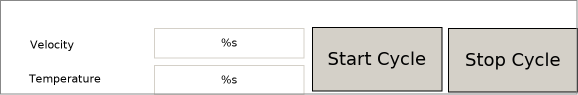
VISUALIZATION BasicHMI  // 578x95
    Textfield (154,28 150x30), "%s", text variable: HMI.Tb_Vel
        OnMouseDown: write HMI.Tb_Vel via VisuDialogs.Numpad
    Label (27,30 120x30), "Velocity"
    Rectangle (312,27 130x64), "Start Cycle"
        tap HMI.Bt_StartCycle
    Label (26,64 120x30), "Temperature"
    Textfield (154,65 150x30), "%s", text variable: HMI.Tb_Temp
        OnMouseDown: write HMI.Tb_Temp via VisuDialogs.Keypad
    Rectangle (448,28 130x64), "Stop Cycle"
        tap HMI.Bt_StopCycle
END_VISUALIZATION

(* stored: Version 1.1.0.1, ProductVersion 3.1.4024.9
   Visu BasicHMI: Id {8b998f78-e1f7-4f21-9e56-fbd1f3cc78cf} *)
